PROGRAM PRG_AlarmHandler
VAR
    fbAlarmManager : FB_AlarmManager;
    bEnableMonitor      : BOOL := TRUE;
    bResetMonitor       : BOOL := FALSE;
    bResetTrigger       : R_TRIG;
    dtCurrentTime       : DT;
    ulSystemTimeMS      : ULINT; // System time in milliseconds (64-bit)
	i : UINT;
END_VAR

// Get current PLC time (simpler approach using system task time)
ulSystemTimeMS := F_GetSystemTime();
// Convert to DATE_AND_TIME using a base date
// Use UDINT to limit to reasonable time range for DT conversion
dtCurrentTime := DT#1970-01-01-00:00 + UDINT_TO_TIME(ULINT_TO_UDINT(ulSystemTimeMS MOD 16#FFFFFFFF));

// Set alarm conditions based on actual system states using alarm IDs
fbAlarmManager.SetAlarmCondition(1001, LinearActuatorPositionUnknown);
fbAlarmManager.SetAlarmCondition(1002, LinearActuatorMotionTimedOut);
fbAlarmManager.SetAlarmCondition(2001, StepperMotorPowerUpFailed);
fbAlarmManager.SetAlarmCondition(2002, StepperMotorHomeOperationFailed);
fbAlarmManager.SetAlarmCondition(2003, StepperMotorHomeOperationInterrupted);
fbAlarmManager.SetAlarmCondition(2004, StepperMotorMotionOperationFailed);
fbAlarmManager.SetAlarmCondition(2005, StepperMotorMotionOperationInterrupted);
fbAlarmManager.SetAlarmCondition(2006, StepperMotorResetOperationFailed);
fbAlarmManager.SetAlarmCondition(9999, EStopEnabled);

fbAlarmManager.Execute();

FOR i := 1 TO MAX_ALARMS DO
    g_AlarmArrayForOPC[i] := AlarmArray[i];
END_FOR

g_nActiveAlarmsOPC := g_nActiveAlarms;
g_nUnackedAlarmsOPC := g_nUnackedAlarms;

// Process acknowledgments from Ignition
IF g_AlarmAckTrigger AND g_AlarmAckRequest > 0 THEN
    fbAlarmManager.AcknowledgeAlarm(g_AlarmAckRequest);
    g_AlarmAckRequest := 0;
    g_AlarmAckTrigger := FALSE;
END_IF

// Handle reset trigger
bResetTrigger(CLK := bResetMonitor);
IF bResetTrigger.Q THEN
	bResetMonitor := FALSE;
END_IF;

END_PROGRAM

(* stored: Version 1.1.0.1, ProductVersion 3.1.4026.11
   POU PRG_AlarmHandler: Id {9a3c7606-d751-41ab-a4a7-f5ba1886e12f}, SpecialFunc None *)
